// TwinCAT 3 PLC project SaftyPLC
// ProgramVersion: 3.1.4026.13
// libraries:
//   Tc2_Standard, * (Beckhoff Automation GmbH)
//   Tc2_System, * (Beckhoff Automation GmbH)
//   Tc2_Utilities, * (Beckhoff Automation GmbH)
//   Tc3_Module, * (Beckhoff Automation GmbH)
// project tree:
//   GVLs/ GVL_IO.TcGVL, GVL_Safety.TcGVL
//   / PlcTask.TcTTO
//   POUs/ MAIN.TcPOU (not stored)

CONFIGURATION SaftyPLC
    RESOURCE PLC ON TwinCAT3
        TASK PlcTask(INTERVAL := T#500us, PRIORITY := 20);
        PROGRAM MAIN WITH PlcTask : MAIN;
    END_RESOURCE
END_CONFIGURATION

// ---- GVLs/GVL_IO.TcGVL

VAR_GLOBAL
	VoltageSet AT%Q*: REAL := 300;
	VoltageAct AT%I*: REAL;
	ControlDrive1121  AT%Q* : UINT;
	StatusDrive1121 AT%I* :UINT;
	ChargingResistor AT%Q* :BOOL;
	up , down : BOOL;
	start  : BOOL := TRUE;
	HwReset: BOOL;
	PowerSupplyReset AT%Q* : BOOL;
END_VAR

// ---- GVLs/GVL_Safety.TcGVL
{attribute 'qualified_only'}
VAR_GLOBAL
	Run			AT%Q* : BOOL := TRUE;
	Start		AT%Q* : BOOL := TRUE;
	Reset		AT%Q* : BOOL;
	
	SafetyInRun	AT%I* : BOOL;
	SaeftyOk 	AT%I* : BOOL;
	
	HWStart		AT%I* : BOOL;
	HWStop		AT%I* : BOOL;
	HWReset		AT%I* : BOOL;
	
	HWerror		AT%Q* : BOOL;
	HWSafetyOk	AT%Q* : BOOL;
	
END_VAR
